{attribute 'qualified_only'}
{attribute 'strict'}
TYPE DeviceLogLevel :
(
	None := 0,
    Verbose,
    Debug,
    Information,
    Warning,
    Error
);
END_TYPE

(* stored: Version 1.1.0.1, ProductVersion 3.1.4024.3
   DUT DeviceLogLevel: Id {ecce11e0-3a86-4cb1-b0dd-06b6944c19f0} *)
